# EPICS substitutions: epics/db/EL3742.substitutions
file "ecSlave.template"
{
  pattern {}
          {}
}
# Oversampling not yet implemented
#file "EL3XXX-chX.template"
#{
#  pattern {CH_ID, LINR,    ESLO,   EOFF,   EGU,        PREC, LOW, LOLO, HIGH, HIHI, HYST, LLSV,       LSV,        HSV,        HHSV      }
#          {1,     "SLOPE", 1,      0,      "DegC",     0,    0,   0,    0,    0,    0,    "NO_ALARM", "NO_ALARM", "NO_ALARM", "NO_ALARM"}
#          {2,     "SLOPE", 1,      0,      "DegC",     0,    0,   0,    0,    0,    0,    "NO_ALARM", "NO_ALARM", "NO_ALARM", "NO_ALARM"}
#}
